DATA_BLOCK "CalcVolume_Tank8_DB"
{ S7_Optimized_Access := 'FALSE' }
VERSION : 0.1
"CalculationVolume"

BEGIN
   IW_Radius := 1.468;
   IW_ValueFromSensor := 18.48597;
   IW_K_for_Tonnag := 1.35;
   IW_K_for_Level := 1.35;
   QW_Volume := 92.65955;
   QW_Tonnag := 125.0904;
   QW_RealLevel := 13.69331;
   sW_S := 6.766776;
   sW_Volume := 92.65955;
   sW_RealLevel := 13.69331;

END_DATA_BLOCK

